{attribute addProperty BoxType "EL1259-0000-0018"}
{attribute addProperty Id "MTO_Inputs_ChannelAT %I*ARRAY[0..7] OF MTO_Inputs_Channel_7DC82D55256320MTI_Inputs_10x_ChannelAT %I*ARRAY[0..84] OF MTI_Inputs_10x_Channel_28B0DBFB43045380MTO_Outputs_10x_ChannelAT %Q*ARRAY[0..84] OF MTO_Outputs_10x_Channel_6165A3A843045380MTI_Outputs_ChannelAT %Q*ARRAY[0..7] OF MTI_Outputs_Channel_DD76C79810961370WcStateAT %I*WcState_98A4DF7520.250InfoDataAT %I*InfoData_0BDED7BF144180"}
{attribute addProperty CRC "3740487018"}
{attribute addProperty SizeInBites "10106"}
{attribute addProperty SizeInBytes "1263.25"}
TYPE EL1259_3504249A :
STRUCT
	{attribute addProperty Name "MTO_Inputs_Channel"}
	MTO_Inputs_Channel : ARRAY[0..7] OF MTO_Inputs_Channel_7DC82D55;
	{attribute addProperty Name "MTI_Inputs_10x_Channel"}
	MTI_Inputs_10x_Channel : ARRAY[0..84] OF MTI_Inputs_10x_Channel_28B0DBFB;
	{attribute addProperty Name "MTO_Outputs_10x_Channel"}
	MTO_Outputs_10x_Channel : ARRAY[0..84] OF MTO_Outputs_10x_Channel_6165A3A8;
	{attribute addProperty Name "MTI_Outputs_Channel"}
	MTI_Outputs_Channel : ARRAY[0..7] OF MTI_Outputs_Channel_DD76C798;
	{attribute addProperty Name "WcState"}
	WcState : WcState_98A4DF75;
	{attribute addProperty Name "InfoData"}
	InfoData : InfoData_0BDED7BF;
END_STRUCT
END_TYPE

(* stored: Version 1.2.0.0, ProductVersion 3.1.4024.9
   DUT EL1259_3504249A: Id {884fb8a8-64a1-4d4f-afce-a7d18783de23} *)
